FUNCTION_BLOCK T_CartesianRobotMaintenanceMode EXTENDS T_NamedBase IMPLEMENTS I_PackMode
VAR
	_cartesianRobot : I_CartesianRobotModule;
END_VAR

METHOD Initialise
VAR_INPUT
	CartesianRobotModule : I_CartesianRobotModule; 
END_VAR
_cartesianRobot := CartesianRobotModule;
END_METHOD

END_FUNCTION_BLOCK

(* stored: Version 1.1.0.1, ProductVersion 3.1.4024.12
   POU T_CartesianRobotMaintenanceMode: Id {a5cf9b46-6efa-499c-9966-a6016ab9e675}, SpecialFunc None
   Method Initialise: Id {6ad3a09a-62bf-4811-84ad-e488e16d2c59} *)
